(* CODESYS project aurel.project

Project tree, tasks and I/O mapping:
  C6_SMART_Single_CAN : C6 SMART ADVANCED, KEB Automation KG, version 3.5.9.70
    application Application
      libraries: Standard, * (System)
      task MainTask (cyclic, interval 8000 µs, priority 0) calls EtherCAT_Master.EtherCAT_Task [EtherCAT_Master.EtherCAT_Task], PLC_PRG
      task PROG1 (cyclic, interval t#16ms, priority 1) calls POU
      program PLC_PRG [ST]
      program POU [LD]
    IoDrvUPS : IoDrvUPS, KEB Automation KG, version 3.5.9.70
        unmapped channels: Power status, 24 Vdc power input status, 24 Vdc power fail counter
    SoftMotion General Drive Pool
    EtherCAT_Master : EtherCAT Master C6 SMART, KEB Automation KG, version 3.5.9.50
      KEB_C6_SMART_Coupler : KEB_C6_SMART_Coupler (3A E-Bus), KEB Automation KG, order no. KEB_C6_SMART_Coupler, version Revision=16#00000003
          settings: DC sync0 cycletime = 8000; DC sync1 cycletime = 8000
        KEBIO_ETHERCAT_DI16_DO16_LS_CoE : KEB_DI16/DO16 1ms LS (00.C6.CB1-1800), KEB Automation KG, order no. KEB_DI16/DO16 LS, version Revision=16#00000001
            settings: DC sync0 cycletime = 8000; DC sync1 cycletime = 8000
            output MOTEUR1 : BIT  // DigitalOutput0
            output MOTEUR2 : BIT  // DigitalOutput1
            input  START : BIT  // DigitalInput0
            input  STOP : BIT  // DigitalInput1
            unmapped channels: DigitalOutput2, DigitalOutput3, DigitalOutput4, DigitalOutput5, DigitalOutput6, DigitalOutput7, DigitalOutput8, DigitalOutput9, DigitalOutput10, DigitalOutput11, DigitalOutput12, DigitalOutput13, DigitalOutput14, DigitalOutput15, DigitalInput2, DigitalInput3, DigitalInput4, DigitalInput5, DigitalInput6, DigitalInput7, DigitalInput8, DigitalInput9, DigitalInput10, DigitalInput11, DigitalInput12, DigitalInput13, DigitalInput14, DigitalInput15
        KEBIO_ETHERCAT_AI4I_CoE : KEB_AI4-I 12 Bit (00.C6.CC1-1300), KEB Automation KG, order no. KEB_AI4-I 12 Bit, version Revision=16#00000001
            settings: DC sync0 cycletime = 8000; DC sync1 cycletime = 8000
            unmapped channels: ResetError, ---, ---, ---, ---, ---, ---, ---, ---, ---, ---, ---, ---, ---, ---, ---, ResetErrorAck, Undervoltage24, EtherCATError, ConfigError, ---, ---, ---, ---, Input0Low, Input1Low, Input2Low, Input3Low, ---, ---, ---, ---, Input0High, Input1High, Input2High, Input3High, ---, ---, ---, ---,
              ---, ---, ---, ---, ---, ---, ---, ---, Input0, Input1, Input2, Input3
        KEBIO_ETHERCAT_AO4U_I : KEB_AO4 16 Bit (00.C6.CC1-1700), KEB Automation KG, order no. KEB_AO4 16 Bit, version Revision=16#00000001
            settings: DC sync0 cycletime = 8000; DC sync1 cycletime = 8000
            unmapped channels: ResetError, ---, ---, ---, ---, ---, ---, ---, ---, ---, ---, ---, ---, ---, ---, ---, AnalogOutput0, AnalogOutput1, AnalogOutput2, AnalogOutput3, ResetErrorAck, Undervoltage, EtherCATError, ConfigError, ---, ---, ---, ---, Output0Overtemp, Output1Overtemp, Output2Overtemp, Output3Overtemp, Output0Open, Output1Open, Output2Open, Output3Open
        KEBIO_ETHERCAT_AI4_PT_NI_TC_CoE : KEB_AI4 Pt/Ni/Thermo 16 Bit (00.C6.CC1-1800), KEB Automation KG, order no. KEB_AI4 Pt/Ni/Thermo 16 Bit, version Revision=16#00000001
            settings: DC sync0 cycletime = 8000; DC sync1 cycletime = 8000
            unmapped channels: ResetError, ---, ---, ---, ---, ---, ---, ---, ---, ---, ---, ---, ---, ---, ---, ---, ResetErrorAck, ---, EtherCATError, ConfigError, ---, ---, ---, ---, Input0Low, Input1Low, Input2Low, Input3Low, ---, ---, ---, ---, Input0High, Input1High, Input2High, Input3High, ---, ---, ---, ---,
              ---, ---, ---, ---, ---, ---, ---, ---, TempInput0, TempInput1, TempInput2, TempInput3
  Configuration
*)

// C6_SMART_Single_CAN/Application/PLC_PRG
PROGRAM PLC_PRG
VAR
END_VAR

END_PROGRAM

// C6_SMART_Single_CAN/Application/POU
PROGRAM POU
VAR
END_VAR

// NETWORK 1

END_PROGRAM
